FUNCTION TryConvert_UDINT_TO_SINT : BOOL
VAR_INPUT
	in : UDINT;
	out : REFERENCE TO SINT;
END_VAR

IF in > DatatypeLimits.MAX_VALUE_OF_UDINT_WHICH_CAN_BE_HELD_IN_A_SINT THEN
	RETURN;
END_IF

out := UDINT_TO_SINT(in);
TryConvert_UDINT_TO_SINT := TRUE;

END_FUNCTION

(* stored: Version 1.1.0.1, ProductVersion 3.1.4024.12
   POU TryConvert_UDINT_TO_SINT: Id {df6f0d19-05ea-41f3-8a17-1cdc47e378d1}, SpecialFunc None *)
